PROGRAM MAIN
VAR
	nAlive: INT;
	breset: BOOL;
	nDemoVariable : INT;
	nCX8200_State	AT %I*	: UINT;
END_VAR

VAR PERSISTENT
	nDemoVar_Persist: INT;
END_VAR

nAlive:= nAlive + 1;
GVL_AHDataModbus.nCX8200_State_MB := nCX8200_State;

P_SystemDK.M_nCyclic(bReset := breset );
P_DALI_DIAG();
DALI_Commissioning();

P_DALI_Energy_Line();

P_AHModbusComm();

//Gange
P_Gang_3_109_Kantine();
P_Gang_4_208();
P_Gang_4_210A();
P_Gang_4_211();

//Foldedøre
P_Foldedoer_4_213();

//Rum
P_Rum_4_206();
P_Rum_4_207();
P_Rum_4_211A();

P_Rum_4_213();
P_Rum_4_215();

P_DigTest();

//P_DALI_Energy_Firmware_Test();

END_PROGRAM

(* stored: Version 1.1.0.1
   POU MAIN: Id {6bf17237-b1a6-4c57-bf47-1238f1ca1a56}, SpecialFunc None *)
